// TIA Portal V20 export
FUNCTION_BLOCK "FB_RealTime"   // FB74, SCL
{ S7_Optimized_Access := 'TRUE' }
// stored: MemoryReserve 100, SetENOAutomatically false
BEGIN
   REGION Description header 
       //==================================================================================
       // POSALUX Swiss SA / (C) Copyright 2024
       //----------------------------------------------------------------------------------
       // Title: FB_RealTime
       // Comment/Function: 
       //
       // Author: Fabien WALDT
       // Engineering: TIA Portal v20
       //----------------------------------------------------------------------------------
       // Change log table:
       // Version  | Date     | Expert in charge | Changes applied
       // ---------|----------|------------------|------------------------------------
       // 00.00.01 | 20260127 | WFA              | First released version
       // ==================================================================================
   END_REGION

   REGION Digital Inputs
       "DB_OPC_RealTime".X_AxisBrakePressCtrl := "DB_DigitalInputs".sX_AxisBrakePressCtrl.sSWStatus;
       "DB_OPC_RealTime".Y_AxisBrakePressCtrl := "DB_DigitalInputs".sY_AxisBrakePressCtrl.sSWStatus;
       "DB_OPC_RealTime".BreakerCtrl := "DB_DigitalInputs".sBreakerCtrl.sSWStatus;
       "DB_OPC_RealTime".CabinetTemperatureCtrl := "DB_DigitalInputs".sCabinetTemperatureCtrl.sSWStatus;
       "DB_OPC_RealTime".UpsPowerFailure := "DB_DigitalInputs".sUPS_PowerFailure.sSWStatus;
       "DB_OPC_RealTime".AirPressureCtrl := "DB_DigitalInputs".sAirPressureCtrl.sSWStatus;
       "DB_OPC_RealTime".ShutterClosed := "DB_DigitalInputs".sShutterClosed.sSWStatus;
       "DB_OPC_RealTime".AirDryerOK := "DB_DigitalInputs".sAirDryerOK.sSWStatus;
       "DB_OPC_RealTime".UPS_BatteryOK := "DB_DigitalInputs".sUPS_BatteryOK.sSWStatus;
       "DB_OPC_RealTime".FrontDoorClosed := "DB_DigitalInputs".sFrontDoorClosed.sSWStatus;
       "DB_OPC_RealTime".InfeedReadyOkStart := "DB_DigitalInputs".sInfeedReadyOK_Start.sSWStatus;
       "DB_OPC_RealTime".CoolingOK := "DB_DigitalInputs".sCoolingOK.sSWStatus;
       "DB_OPC_RealTime".PowerReady := "DB_DigitalInputs".sPowerReady.sSWStatus;
       "DB_OPC_RealTime".AlarmI2T := "DB_DigitalInputs".sAlarmI2T.sSWStatus;
       "DB_OPC_RealTime".HeadLaserBusy := "DB_DigitalInputs".sHeadLaserBusy.sSWStatus;
       "DB_OPC_RealTime".HeadLaserBreaker := "DB_DigitalInputs".sHeadLaserBreaker.sSWStatus;
       "DB_OPC_RealTime".FrontDoorLocked := "DB_DigitalInputs".sFrontDoorLocked.sSWStatus;
       "DB_OPC_RealTime".UPS_CommonAlarm := "DB_DigitalInputs".sUPS_CommonAlarm.sSWStatus;
       "DB_OPC_RealTime".UPS_BatteryLow := "DB_DigitalInputs".sUPS_BatteryLow.sSWStatus;
       "DB_OPC_RealTime".HeadChillerHighPressure := "DB_DigitalInputs".sHeadChillerHighPressure.sSWStatus;
       "DB_OPC_RealTime".HeadChillerWaterTemperature := "DB_DigitalInputs".sHeadChillerWaterTemperature.sSWStatus;
       "DB_OPC_RealTime".HeadChillerFlow := "DB_DigitalInputs".sHeadChillerFlow.sSWStatus;
       "DB_OPC_RealTime".HeadChillerCollectivFault := "DB_DigitalInputs".sHeadChillerCollectivFault.sSWStatus;
       "DB_OPC_RealTime".HeadChillerWaterLevel := "DB_DigitalInputs".sHeadChillerWaterLevel.sSWStatus;
       "DB_OPC_RealTime".UpsByPassActive := "DB_DigitalInputs".sUPS_ByPassActive.sSWStatus;
       "DB_OPC_RealTime".HeadChillerAmbiantTemperature := "DB_DigitalInputs".sHeadChillerAmbiantTemperature.sSWStatus;
       "DB_OPC_RealTime".LoadClampOpened := "DB_DigitalInputs".sLoadClampOpened.sSWStatus;
       "DB_OPC_RealTime".LoadClampNotClosedWithPart := "DB_DigitalInputs".sLoadClampNotClosedWithPart.sSWStatus;
       "DB_OPC_RealTime".UnloadClampOpened := "DB_DigitalInputs".sUnloadClampOpened.sSWStatus;
       "DB_OPC_RealTime".UpsFault := "DB_DigitalInputs".sUPS_Fault.sSWStatus;
       "DB_OPC_RealTime".InternalGateLocked := "DB_DigitalInputs".sInternalGateLocked.sSWStatus;
       "DB_OPC_RealTime".ExternalGateLocked := "DB_DigitalInputs".sExternalGateLocked.sSWStatus;
       "DB_OPC_RealTime".InverterActive := "DB_DigitalInputs".sInverterActive.sSWStatus;
       "DB_OPC_RealTime".UnloadClampNotClosedWithPart := "DB_DigitalInputs".sUnloadClampNotClosedWithPart.sSWStatus;
       "DB_OPC_RealTime".InternalGateOpened := "DB_DigitalInputs".sInternalGateOpened.sSWStatus;
       "DB_OPC_RealTime".ExternalGateOpened := "DB_DigitalInputs".sExternalGateOpened.sSWStatus;
       "DB_OPC_RealTime".PowerMeterBackCtrl := "DB_DigitalInputs".sPowerMeterBackCtrl.sSWStatus;
       "DB_OPC_RealTime".PowerMeterFrontCtrl := "DB_DigitalInputs".sPowerMeterFrontCtrl.sSWStatus;
       "DB_OPC_RealTime".HeadChillerCutOff := "DB_DigitalInputs".sHeadChillerCutOff.sSWStatus;
       "DB_OPC_RealTime".HeadChillerTemperature := "DB_DigitalInputs".sHeadChillerTemperature.sSWStatus;
       "DB_OPC_RealTime".ClampingOpenCtrl := "DB_DigitalInputs".sClampingOpenCtrl.sSWStatus;
       "DB_OPC_RealTime".B_AxisBrakeReleasedCtrl := "DB_DigitalInputs".sB_Axis_BrakeReleasedCtrl.sSWStatus;
       "DB_OPC_RealTime".B_AxisReferencePoint := "DB_DigitalInputs".sB_AxisReferencePoint.sSWStatus;
       "DB_OPC_RealTime".SourceChillerHighPressure := "DB_DigitalInputs".sSourceChillerHighPressure.sSWStatus;
       "DB_OPC_RealTime".SourceChillerWaterTemperature := "DB_DigitalInputs".sSourceChillerWaterTemperature.sSWStatus;
       "DB_OPC_RealTime".SourceChillerFlow := "DB_DigitalInputs".sSourceChillerFlow.sSWStatus;
       "DB_OPC_RealTime".SourceChillerCollectivFault := "DB_DigitalInputs".sSourceChillerCollectivFault.sSWStatus;
       "DB_OPC_RealTime".SourceChillerWaterLevel := "DB_DigitalInputs".sSourceChillerWaterLevel.sSWStatus;
       "DB_OPC_RealTime".SourceChillerAmbiantTemperature := "DB_DigitalInputs".sSourceChillerAmbiantTemperature.sSWStatus;
       "DB_OPC_RealTime".SourceChillerCutOff := "DB_DigitalInputs".sSourceChillerCutOff.sSWStatus;
       "DB_OPC_RealTime".SourceChillerTemperature := "DB_DigitalInputs".sSourceChillerTemperature.sSWStatus;
   END_REGION

   REGION Digital Outputs
       "DB_OPC_RealTime".OperatingCounter := "DB_DigitalOutputs".sOperatingCounter.sSWStatus;
       "DB_OPC_RealTime".GeneralAirValve := "DB_DigitalOutputs".sGeneralAirValve.sSWStatus;
       "DB_OPC_RealTime".SmartLineDisable := "DB_DigitalOutputs".sSmartLineDisable.sSWStatus;
       "DB_OPC_RealTime".MachineLight := "DB_DigitalOutputs".sMachineLight.sSWStatus;
       "DB_OPC_RealTime".MachineLightBack := "DB_DigitalOutputs".sMachineLightBack.sSWStatus;
       "DB_OPC_RealTime".LightTowerOrange := "DB_DigitalOutputs".sLightTowerOrange.sSWStatus;
       "DB_OPC_RealTime".LightTowerRed := "DB_DigitalOutputs".sLightTowerRed.sSWStatus;
       "DB_OPC_RealTime".LightTowerBlue := "DB_DigitalOutputs".sLightTowerBlue.sSWStatus;
       "DB_OPC_RealTime".LightTowerGreen := "DB_DigitalOutputs".sLightTowerGreen.sSWStatus;
       "DB_OPC_RealTime".LightTowerWhite := "DB_DigitalOutputs".sLightTowerWhite.sSWStatus;
       "DB_OPC_RealTime".Backlight := "DB_DigitalOutputs".sBacklight.sSWStatus;
       "DB_OPC_RealTime".InfeedON := "DB_DigitalOutputs".sInfeedON.sSWStatus;
       "DB_OPC_RealTime".AxisActivation := "DB_DigitalOutputs".sAxisActivation.sSWStatus;
       "DB_OPC_RealTime".BuzzerActivation := "DB_DigitalOutputs".sBuzzerActivation.sSWStatus;
       "DB_OPC_RealTime".ElbaronPowerON := "DB_DigitalOutputs".sElbaronPowerON.sSWStatus;
       "DB_OPC_RealTime".ObservationCameraLight := "DB_DigitalOutputs".sObservationCameraLight.sSWStatus;
       "DB_OPC_RealTime".LaserExternalDoorOpening := "DB_DigitalOutputs".sLaserExternalDoorOpening.sSWStatus;
       "DB_OPC_RealTime".CoolingStart := "DB_DigitalOutputs".sCoolingStart.sSWStatus;
       "DB_OPC_RealTime".X_AxisBrakeActivation := "DB_DigitalOutputs".sX_AxisBrakeActivation.sSWStatus;
       "DB_OPC_RealTime".Y_AxisBrakeActivation := "DB_DigitalOutputs".sY_AxisBrakeActivation.sSWStatus;
       "DB_OPC_RealTime".AxisB_TeachInClampingPart := "DB_DigitalOutputs".sAxisB_TeachInClampingPart.sSWStatus;
       "DB_OPC_RealTime".EPO_UPS := "DB_DigitalOutputs".sEPO_UPS.sSWStatus;
       "DB_OPC_RealTime".HeadLaserStart := "DB_DigitalOutputs".sHeadLaserStart.sSWStatus;
       "DB_OPC_RealTime".HeadLaserStop := "DB_DigitalOutputs".sHeadLaserStop.sSWStatus;
       "DB_OPC_RealTime".Axis2_PowerContactor := "DB_DigitalOutputs".sAxis2_PowerContactor.sSWStatus;
       "DB_OPC_RealTime".GasAssistOn := "DB_DigitalOutputs".sGasAssistOn.sSWStatus;
       "DB_OPC_RealTime".SmartLineReset := "DB_DigitalOutputs".sSmartLineReset.sSWStatus;
       "DB_OPC_RealTime".XY_AxisPowerContactor := "DB_DigitalOutputs".sXY_AxisPowerContactor.sSWStatus;
       "DB_OPC_RealTime".LaserAirPressureProcess := "DB_DigitalOutputs".sLaserAirPressureProcess.sSWStatus;
       "DB_OPC_RealTime".Bus60V_PowerContactor := "DB_DigitalOutputs".sBus60V_PowerContactor.sSWStatus;
       "DB_OPC_RealTime".LoadClampClosing := "DB_DigitalOutputs".sLoadClampClosing.sSWStatus;
       "DB_OPC_RealTime".LoadClampOpening := "DB_DigitalOutputs".sLoadClampOpening.sSWStatus;
       "DB_OPC_RealTime".UnloadClampClosing := "DB_DigitalOutputs".sUnloadClampClosing.sSWStatus;
       "DB_OPC_RealTime".UnloadClampOpening := "DB_DigitalOutputs".sUnloadClampOpening.sSWStatus;
       "DB_OPC_RealTime".ClampingOpening := "DB_DigitalOutputs".sClampingOpening.sSWStatus;
       "DB_OPC_RealTime".ClampingClosing := "DB_DigitalOutputs".sClampingClosing.sSWStatus;
       "DB_OPC_RealTime".B_AxisBrakeRelease := "DB_DigitalOutputs".sB_AxisBrakeRelease.sSWStatus;
       "DB_OPC_RealTime".Suction := "DB_DigitalOutputs".sSuction.sSWStatus;
       "DB_OPC_RealTime".ExternalGateClosing := "DB_DigitalOutputs".sExternalGateClosing.sSWStatus;
       "DB_OPC_RealTime".ExternalGateOpening := "DB_DigitalOutputs".sExternalGateOpening.sSWStatus;
       "DB_OPC_RealTime".InternalGateClosing := "DB_DigitalOutputs".sInternalGateClosing.sSWStatus;
       "DB_OPC_RealTime".InternalGateOpening := "DB_DigitalOutputs".sInternalGateOpening.sSWStatus;
       "DB_OPC_RealTime".PowerMeterRetract := "DB_DigitalOutputs".sPowerMeterRetract.sSWStatus;
       "DB_OPC_RealTime".PowerMeterAdvance := "DB_DigitalOutputs".sPowerMeterAdvance.sSWStatus;
       "DB_OPC_RealTime".Blowing := "DB_DigitalOutputs".sBlowing.sSWStatus;
   END_REGION

   REGION Analog Inputs
       "DB_OPC_RealTime".LaserPowerMeter := "DB_AnalogInputs".sLaserPowerMeter.sSWRealValue;
       "DB_OPC_RealTime".AxisB_ClampingPart := "DB_AnalogInputs".sAxisB_ClampingPart.sSWRealValue;
       "DB_OPC_RealTime".LaserAirPressureProcess_1 := "DB_AnalogInputs".sLaserAirPressureProcess.sSWRealValue;
       "DB_OPC_RealTime".InletAirPressure := "DB_AnalogInputs".sInletAirPressure.sSWRealValue;
       "DB_OPC_RealTime".AmbiantTemperature := "DB_AnalogInputs".sAmbiantTemperature.sSWRealValue;
       "DB_OPC_RealTime".MachineTemperature := "DB_AnalogInputs".sMachineTemperature.sSWRealValue;
       "DB_OPC_RealTime".Cold_WaterTemperatureInput := "DB_AnalogInputs".sCold_WaterTemperatureInput.sSWRealValue;
       "DB_OPC_RealTime".Cold_WaterTemperatureOutput := "DB_AnalogInputs".sCold_WaterTemperatureOutput.sSWRealValue;
       "DB_OPC_RealTime".X_AxisTemperaturePT1000 := "DB_AnalogInputs".sX_AxisTemperaturePT1000.sSWRealValue;
       "DB_OPC_RealTime".Y_AxisTemperaturePT1000 := "DB_AnalogInputs".sY_AxisTemperaturePT1000.sSWRealValue;
       "DB_OPC_RealTime".X_AxisTemperaturePTC := "DB_AnalogInputs".sX_AxisTemperaturePTC.sSWRealValue;
       "DB_OPC_RealTime".Y_AxisTemperaturePTC := "DB_AnalogInputs".sY_AxisTemperaturePTC.sSWRealValue;
       "DB_OPC_RealTime".NozzleOverpressure := "DB_AnalogInputs".sNozzleOverpressure.sSWRealValue;
       "DB_OPC_RealTime".OpticalPathOverpressure := "DB_AnalogInputs".sOpticalPathOverpressure.sSWRealValue;
       "DB_OPC_RealTime".LaserHeadOverpressure := "DB_AnalogInputs".sLaserHeadOverpressure.sSWRealValue;
       "DB_OPC_RealTime".ZLAxisOverpressure := "DB_AnalogInputs".sZLAxisOverpressure.sSWRealValue;
       "DB_OPC_RealTime".XYAxisOverpressure := "DB_AnalogInputs".sXYAxisOverpressure.sSWRealValue;
       "DB_OPC_RealTime".LeftAspiration := "DB_AnalogInputs".sLeftAspiration.sSWRealValue;
       "DB_OPC_RealTime".RightAspiration := "DB_AnalogInputs".sRightAspiration.sSWRealValue;
       "DB_OPC_RealTime".ClimTemperature := "DB_AnalogInputs".sClimTemperature.sSWRealValue;
       "DB_OPC_RealTime".SensorControllerStation1 := "DB_AnalogInputs".sSensorControllerStation1.sSWRealValue;
       "DB_OPC_RealTime".CabinetTemperature := "DB_AnalogInputs".sCabinetTemperature.sSWRealValue;
   END_REGION

   REGION Analog Outputs
       "DB_OPC_RealTime".NozzleOverpressureSetPoint := "DB_AnalogOutputs".sNozzleOverpressureSetPoint.sSWRealValue;
       "DB_OPC_RealTime".VentilatorSetPoint := "DB_AnalogOutputs".sVentilatorSetPoint.sSWRealValue;
       "DB_OPC_RealTime".PropValveClimSetPoint := "DB_AnalogOutputs".sPropValveClimSetPoint.sSWRealValue;
   END_REGION
END_FUNCTION_BLOCK
